TYPE TYP_ALARM_DEVICE_CONFIG :
STRUCT
	Name : STRING;
	Handler : REFERENCE TO FB_ALARM_HANDLER;
END_STRUCT
END_TYPE

(* stored: Version 1.1.0.1, ProductVersion 3.1.4024.12
   DUT TYP_ALARM_DEVICE_CONFIG: Id {cd00d540-27a1-4eb4-960e-869cca3352d6} *)
